FUNCTION_BLOCK FB_RFTRIG
VAR_INPUT
	// signal to detect
	CLK:	BOOL;
END_VAR
VAR_OUTPUT
	Q: BOOL;
END_VAR
VAR
	ftrig:	F_TRIG;
	rtrig:	R_TRIG;
END_VAR

ftrig(CLK:=CLK);
rtrig(CLK:=CLK);
Q := ftrig.Q OR rtrig.Q;

END_FUNCTION_BLOCK

(* stored: Version 1.1.0.1, ProductVersion 3.1.4024.9
   POU FB_RFTRIG: Id {4f47cf7f-076d-4104-944c-d0158381e70f}, SpecialFunc None *)
